FUNCTION_BLOCK PUBLISH_1
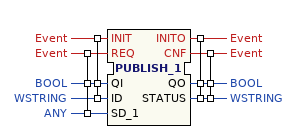
  EVENT_INPUT
    INIT WITH QI, ID;
    REQ WITH QI, SD_1;
  END_EVENT
  EVENT_OUTPUT
    INITO WITH QO, STATUS;
    CNF WITH QO, STATUS;
  END_EVENT
  VAR_INPUT
    QI : BOOL;
    ID : WSTRING;
    SD_1 : ANY;
  END_VAR
  VAR_OUTPUT
    QO : BOOL;
    STATUS : WSTRING;
  END_VAR
END_FUNCTION_BLOCK
